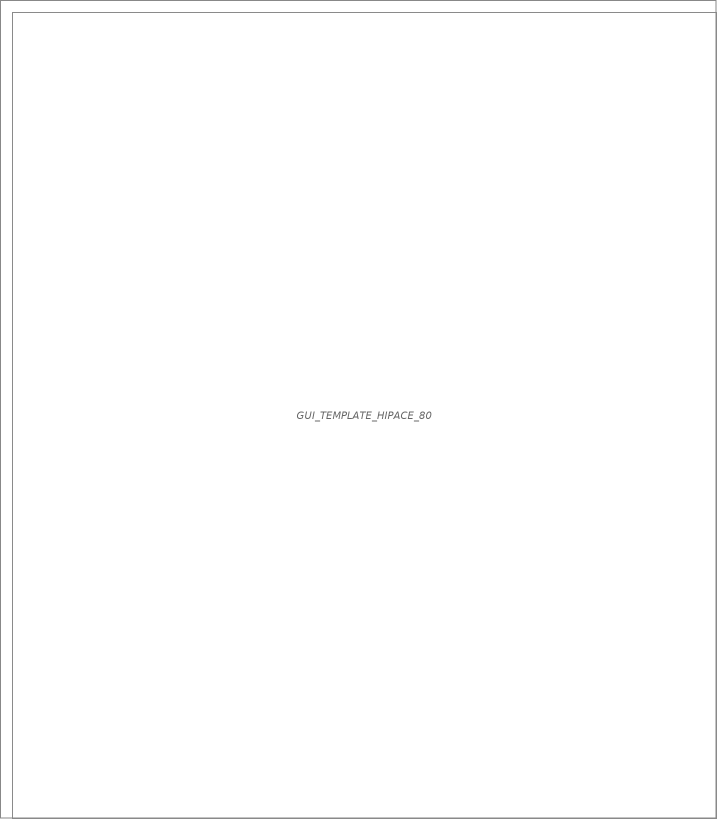
VISUALIZATION VISU_NOTT_TP  // 717x819
    Frame (12,12 705x807)
        shows GUI_TEMPLATE_HIPACE_80(m_Instance := MAIN.nott_cryo_ctrl.evac.pump_tmp)
END_VISUALIZATION

(* stored: Version 1.1.0.1, ProductVersion 3.1.4026.18
   Visu VISU_NOTT_TP: Id {a1e68670-4ed7-4f7c-a510-b68c72f28499} *)
